// Mitsubishi GX Developer project: Solution   PLC: FX1S

PROGRAM MAIN
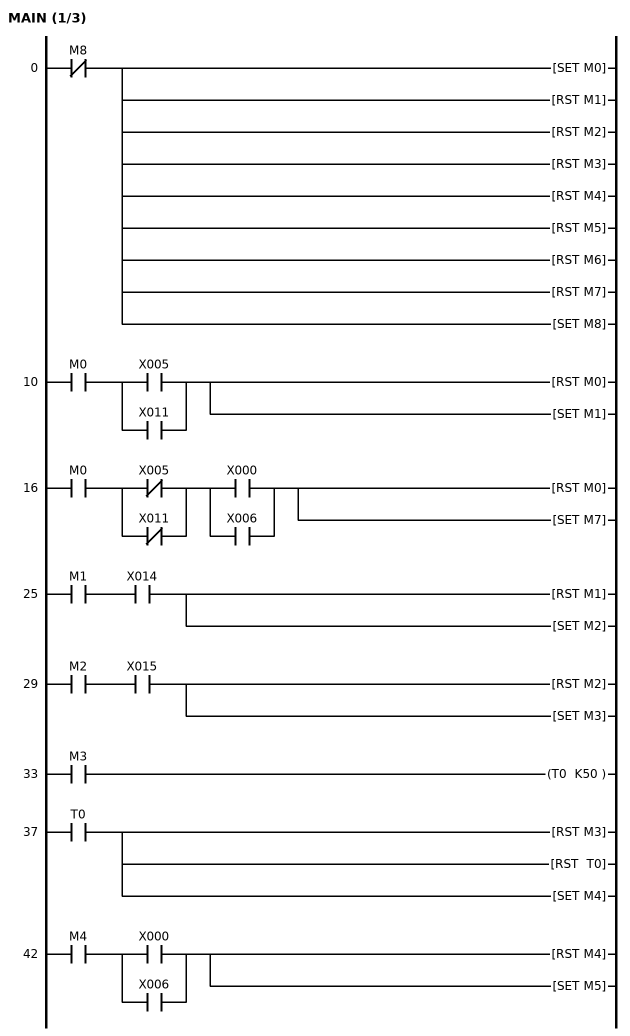
0     LDI     M8
      SET     M0
      RST     M1
      RST     M2
      RST     M3
      RST     M4
      RST     M5
      RST     M6
      RST     M7
      SET     M8
10    LD      M0
      LD      X005
      OR      X011
      ANB
      RST     M0
      SET     M1
16    LD      M0
      LDI     X005
      ORI     X011
      ANB
      LD      X000
      OR      X006
      ANB
      RST     M0
      SET     M7
25    LD      M1
      AND     X014
      RST     M1
      SET     M2
29    LD      M2
      AND     X015
      RST     M2
      SET     M3
33    LD      M3
      OUT     T0 K50
37    LD      T0
      RST     M3
      RST     T0
      SET     M4
42    LD      M4
      LD      X000
      OR      X006
      ANB
      RST     M4
      SET     M5
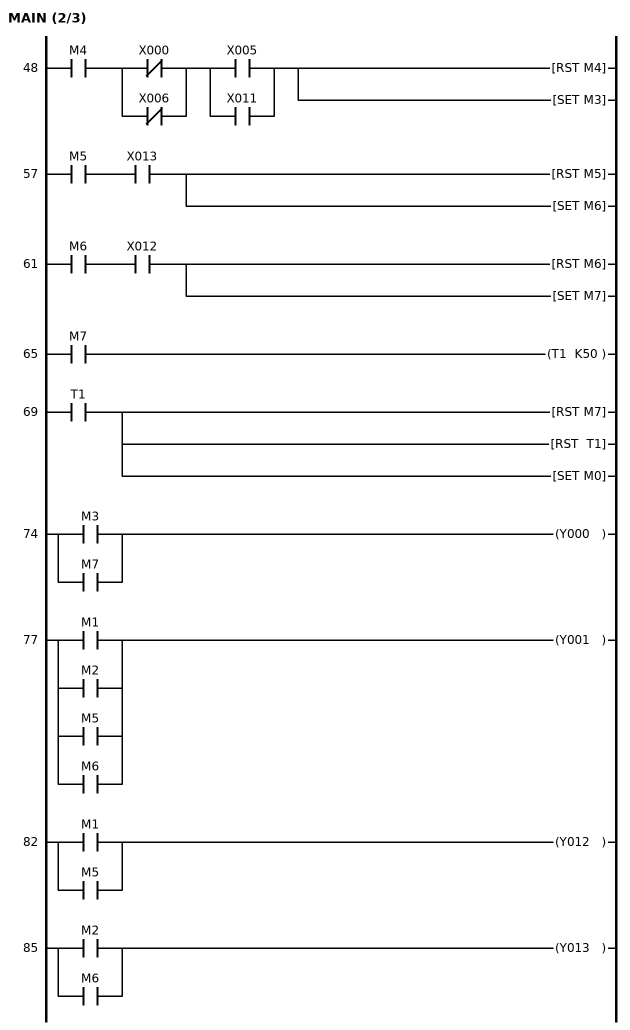
48    LD      M4
      LDI     X000
      ORI     X006
      ANB
      LD      X005
      OR      X011
      ANB
      RST     M4
      SET     M3
57    LD      M5
      AND     X013
      RST     M5
      SET     M6
61    LD      M6
      AND     X012
      RST     M6
      SET     M7
65    LD      M7
      OUT     T1 K50
69    LD      T1
      RST     M7
      RST     T1
      SET     M0
74    LD      M3
      OR      M7
      OUT     Y000
77    LD      M1
      OR      M2
      OR      M5
      OR      M6
      OUT     Y001
82    LD      M1
      OR      M5
      OUT     Y012
85    LD      M2
      OR      M6
      OUT     Y013
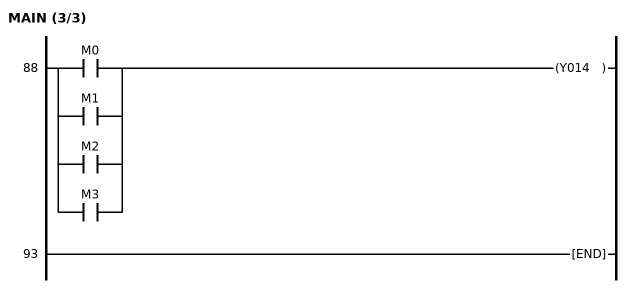
88    LD      M0
      OR      M1
      OR      M2
      OR      M3
      OUT     Y014
93    END
END_PROGRAM
